// SIMATIC S7-200 SMART project (STEP 7-Micro/WIN SMART), CPU ST40

SYMBOL_TABLE Table 1
Start_SW         I0.0
Stop_SW          I0.1
Memory           M0.0
Timer            T101
Motor            Q0.0
END_SYMBOL_TABLE

ORGANIZATION_BLOCK MAIN:OB1
TITLE=Program Comments
BEGIN
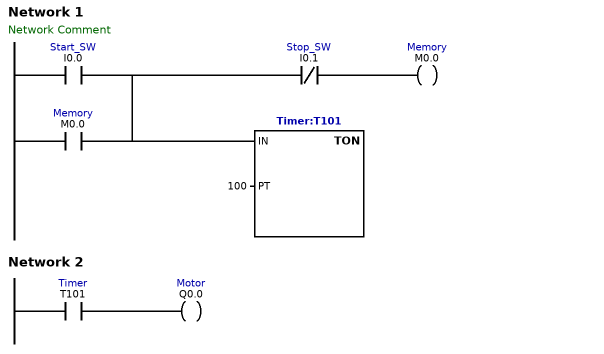
Network 1
// Network Comment
// (network saved uncompiled; LAD cells follow)
// row 0: c0 -| |- Start_SW:I0.0 v  c1 --  c2 -|/|- Stop_SW:I0.1  c3 -( ) Memory:M0.0
// row 1: c0 -| |- Memory:M0.0 ^  c1 --  c2 [TON Timer:T101 IN:=power@row1, PT:=100]
// row 2: c2 [box]
Network 2
// (network saved uncompiled; LAD cells follow)
// row 0: c0 -| |- Timer:T101  c1 -( ) Motor:Q0.0
END_ORGANIZATION_BLOCK
